// Mitsubishi GX Works2 project: z07   PLC: Q02/Q02H

PROGRAM MAIN
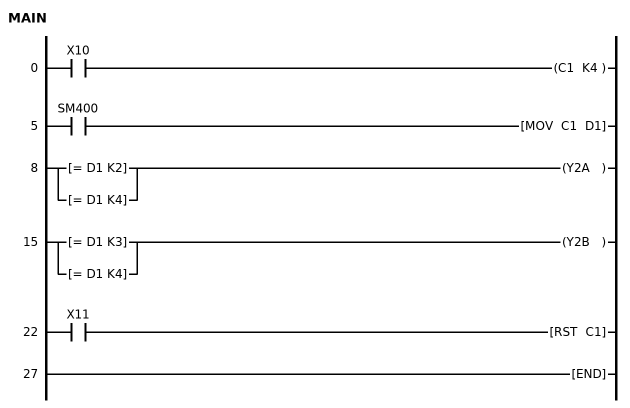
0     LD      X10
      OUT     C1 K4
5     LD      SM400
      MOV     C1 D1
8     LD=     D1 K2
      OR=     D1 K4
      OUT     Y2A
15    LD=     D1 K3
      OR=     D1 K4
      OUT     Y2B
22    LD      X11
      RST     C1
27    END
END_PROGRAM
